Staubli VAL3: slot.pgx

public program slot(event& event_)
begin
  switch event_.nType
    case EV:DRY_RUN
      call setDryRunSig(event_.sParam=="1")
    break
    case EV:START_COMPLETE
      SYS:doSecu[0]=true
    SYS:doSecu[1]=true
    break
  endSwitch
end
